# EPICS substitutions: apps/caenHvApp/Db/sums/HVDC_sums.substitutions
file "db/HVDC_sums.db" {
    pattern {S,R,L}
    {"1","1","1"}
    {"1","1","2"}
    {"1","2","1"}
    {"1","2","2"}
    {"1","3","1"}
    {"1","3","2"}
    {"2","1","1"}
    {"2","1","2"}
    {"2","2","1"}
    {"2","2","2"}
    {"2","3","1"}
    {"2","3","2"}
    {"3","1","1"}
    {"3","1","2"}
    {"3","2","1"}
    {"3","2","2"}
    {"3","3","1"}
    {"3","3","2"}
    {"4","1","1"}
    {"4","1","2"}
    {"4","2","1"}
    {"4","2","2"}
    {"4","3","1"}
    {"4","3","2"}
    {"5","1","1"}
    {"5","1","2"}
    {"5","2","1"}
    {"5","2","2"}
    {"5","3","1"}
    {"5","3","2"}
    {"6","1","1"}
    {"6","1","2"}
    {"6","2","1"}
    {"6","2","2"}
    {"6","3","1"}
    {"6","3","2"}
}
